// TIA Portal project "2022.10.19_FB_视觉分拣" (V17)
// Vorlageprojekt für das Buch mit Zielsystem S7-1200

(* hardware
DEVICE "S7-1200-Station_1"  S7-1200 Station
   slot 0: "Baugruppenträger_0"  Rack  V1.0
   slot 1: "PLC_1"  CPU 1214C DC/DC/Rly  6ES7 214-1HG40-0XB0  V4.5
*)

// ===== PLC "PLC_1"  CPU 1214C DC/DC/Rly =====

VAR_GLOBAL   // PLC tag table "XML 中的变量表_1"
   "启动按钮" AT %I0.0 : Bool;
   "停止按钮" AT %I0.1 : Bool;
   "复位信号" AT %Q0.2 : Bool;
   "急停" AT %I0.3 : Bool;
   "左电传感器" AT %I0.5 : Bool;
   "后电传感器" AT %I0.7 : Bool;
   "手动模式" AT %I1.0 : Bool;
   "自动模式" AT %I1.1 : Bool;
   "启动指示灯" AT %Q0.0 : Bool;
   "停止指示灯" AT %Q0.1 : Bool;
   "送料带" AT %Q0.3 : Bool;
   "直行电机" AT %Q0.4 : Bool;
   "左换向" AT %Q0.5 : Bool;
   "右换向" AT %Q0.6 : Bool;
   "后1带—原料" AT %Q0.7 : Bool;
   "右1带—基座" AT %Q1.0 : Bool;
   "左1带_产品盖" AT %Q1.1 : Bool;
   "出料台" AT %Q1.2 : Bool;
   "挡板" AT %Q1.3 : Bool;
   "视觉相机" AT %ID30 : DWord;
   "右电传感器" AT %I0.6 : Bool;
END_VAR

DATA_BLOCK "主程序DB"   // DB1
{ S7_Optimized_Access := 'TRUE' }
VERSION : 0.1
   VAR
      核心分拣区程序步 : Int;
   END_VAR
BEGIN
END_DATA_BLOCK

DATA_BLOCK "视觉核心分拣区FB块_DB"   // DB3
{ S7_Optimized_Access := 'TRUE' }
VERSION : 0.1
// stored: InstanceOfName 视觉核心分拣区FB块
"视觉核心分拣区FB块"
BEGIN
END_DATA_BLOCK

FUNCTION_BLOCK "视觉核心分拣区FB块"   // FB1, LAD
{ S7_Optimized_Access := 'TRUE' }
VERSION : 0.1
   VAR_INPUT
      视觉相机数据 : DWord;
      后电传感器 : Bool;
      左电传感器 : Bool;
      右电传感器 : Bool;
   END_VAR
   VAR_OUTPUT
      直行电机 : Bool;
      左转向 : Bool;
      右转向 : Bool;
   END_VAR
   VAR_IN_OUT
      程序步 : Int;
   END_VAR
   VAR
      中间变量1 : Bool;
      中间变量2 : Bool;
      中间变量3 : Bool;
   END_VAR
   VAR_TEMP   // added for the SCL form of the ladder/FBD networks
      _w1 : Bool;
   END_VAR
BEGIN

REGION Network 1: 物料判断
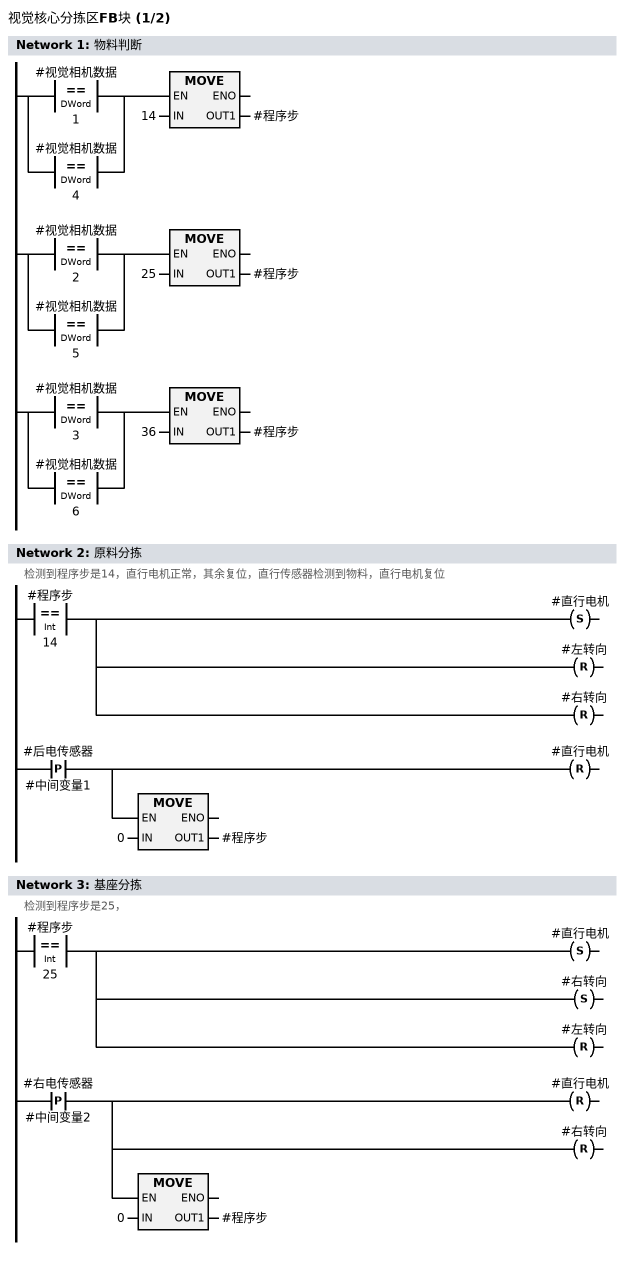
   RUNG wire#powerrail
      { S7_Templates := "SrcType := DWord" } EQ_Contact(in1 := #视觉相机数据, in2 := 1)
      wire#w1
      Move(in := 14, out1 => #程序步)
   END_RUNG
   RUNG wire#powerrail
      { S7_Templates := "SrcType := DWord" } EQ_Contact(in1 := #视觉相机数据, in2 := 4)
   END_RUNG wire#w1
   RUNG wire#powerrail
      { S7_Templates := "SrcType := DWord" } EQ_Contact(in1 := #视觉相机数据, in2 := 2)
      wire#w2
      Move(in := 25, out1 => #程序步)
   END_RUNG
   RUNG wire#powerrail
      { S7_Templates := "SrcType := DWord" } EQ_Contact(in1 := #视觉相机数据, in2 := 5)
   END_RUNG wire#w2
   RUNG wire#powerrail
      { S7_Templates := "SrcType := DWord" } EQ_Contact(in1 := #视觉相机数据, in2 := 3)
      wire#w3
      Move(in := 36, out1 => #程序步)
   END_RUNG
   RUNG wire#powerrail
      { S7_Templates := "SrcType := DWord" } EQ_Contact(in1 := #视觉相机数据, in2 := 6)
   END_RUNG wire#w3
   // the same network as SCL:
   IF (#视觉相机数据 = 1) OR (#视觉相机数据 = 4) THEN #程序步 := 14; END_IF;
   IF (#视觉相机数据 = 2) OR (#视觉相机数据 = 5) THEN #程序步 := 25; END_IF;
   IF (#视觉相机数据 = 3) OR (#视觉相机数据 = 6) THEN #程序步 := 36; END_IF;
END_REGION

REGION Network 2: 原料分拣
   // 检测到程序步是14，直行电机正常，其余复位，直行传感器检测到物料，直行电机复位
   RUNG wire#powerrail
      { S7_Templates := "SrcType := Int" } EQ_Contact(in1 := #程序步, in2 := 14)
      wire#w1
      S_Coil( #直行电机 )
   END_RUNG
   RUNG wire#w1
      R_Coil( #左转向 )
   END_RUNG
   RUNG wire#w1
      R_Coil( #右转向 )
   END_RUNG
   RUNG wire#powerrail
      P_Contact(operand := #后电传感器, bit := #中间变量1)
      wire#w2
      R_Coil( #直行电机 )
   END_RUNG
   RUNG wire#w2
      Move(in := 0, out1 => #程序步)
   END_RUNG
   // the same network as SCL:
   IF #程序步 = 14 THEN
       #直行电机 := TRUE;
       #左转向 := FALSE;
       #右转向 := FALSE;
   END_IF;
   #_w1 := #后电传感器 AND NOT #中间变量1;   // rising edge of #后电传感器
   #中间变量1 := #后电传感器;
   IF #_w1 THEN
       #直行电机 := FALSE;
       #程序步 := 0;
   END_IF;
END_REGION

REGION Network 3: 基座分拣
   // 检测到程序步是25，
   RUNG wire#powerrail
      { S7_Templates := "SrcType := Int" } EQ_Contact(in1 := #程序步, in2 := 25)
      wire#w1
      S_Coil( #直行电机 )
   END_RUNG
   RUNG wire#w1
      S_Coil( #右转向 )
   END_RUNG
   RUNG wire#w1
      R_Coil( #左转向 )
   END_RUNG
   RUNG wire#powerrail
      P_Contact(operand := #右电传感器, bit := #中间变量2)
      wire#w2
      R_Coil( #直行电机 )
   END_RUNG
   RUNG wire#w2
      R_Coil( #右转向 )
   END_RUNG
   RUNG wire#w2
      Move(in := 0, out1 => #程序步)
   END_RUNG
   // the same network as SCL:
   IF #程序步 = 25 THEN
       #直行电机 := TRUE;
       #右转向 := TRUE;
       #左转向 := FALSE;
   END_IF;
   #_w1 := #右电传感器 AND NOT #中间变量2;   // rising edge of #右电传感器
   #中间变量2 := #右电传感器;
   IF #_w1 THEN
       #直行电机 := FALSE;
       #右转向 := FALSE;
       #程序步 := 0;
   END_IF;
END_REGION

REGION Network 4: 基盖
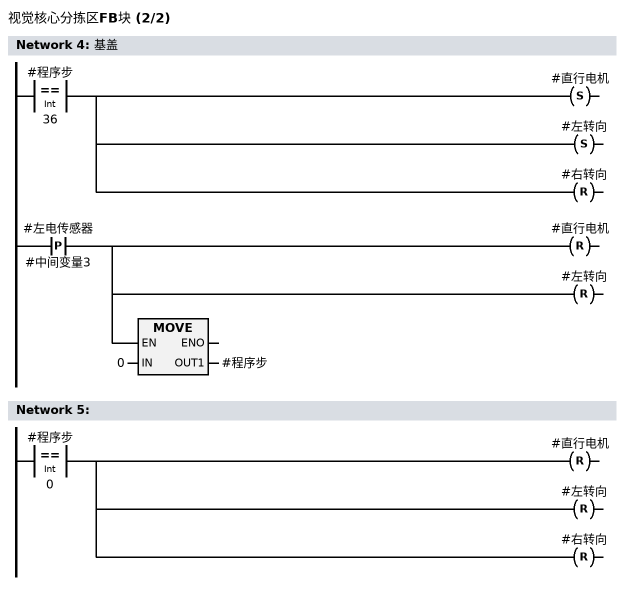
   RUNG wire#powerrail
      { S7_Templates := "SrcType := Int" } EQ_Contact(in1 := #程序步, in2 := 36)
      wire#w1
      S_Coil( #直行电机 )
   END_RUNG
   RUNG wire#w1
      S_Coil( #左转向 )
   END_RUNG
   RUNG wire#w1
      R_Coil( #右转向 )
   END_RUNG
   RUNG wire#powerrail
      P_Contact(operand := #左电传感器, bit := #中间变量3)
      wire#w2
      R_Coil( #直行电机 )
   END_RUNG
   RUNG wire#w2
      R_Coil( #左转向 )
   END_RUNG
   RUNG wire#w2
      Move(in := 0, out1 => #程序步)
   END_RUNG
   // the same network as SCL:
   IF #程序步 = 36 THEN
       #直行电机 := TRUE;
       #左转向 := TRUE;
       #右转向 := FALSE;
   END_IF;
   #_w1 := #左电传感器 AND NOT #中间变量3;   // rising edge of #左电传感器
   #中间变量3 := #左电传感器;
   IF #_w1 THEN
       #直行电机 := FALSE;
       #左转向 := FALSE;
       #程序步 := 0;
   END_IF;
END_REGION

REGION Network 5
   RUNG wire#powerrail
      { S7_Templates := "SrcType := Int" } EQ_Contact(in1 := #程序步, in2 := 0)
      wire#w1
      R_Coil( #直行电机 )
   END_RUNG
   RUNG wire#w1
      R_Coil( #左转向 )
   END_RUNG
   RUNG wire#w1
      R_Coil( #右转向 )
   END_RUNG
   // the same network as SCL:
   IF #程序步 = 0 THEN
       #直行电机 := FALSE;
       #左转向 := FALSE;
       #右转向 := FALSE;
   END_IF;
END_REGION
END_FUNCTION_BLOCK

FUNCTION "MHJ-PLC-Lab-Function-S71200" : Void   // FC9000, SCL
{ S7_Optimized_Access := 'TRUE' }
VERSION : 0.1
   VAR_TEMP
      rdTimeReturn : Int;
      outputTime : DTL;
      SyncVal : Byte;
      forVal : Int;
      forVal_2 : Int;
      Value : Byte;
   END_VAR
   VAR CONSTANT
      CompVal : Byte := 16#34;
      Value_01 : Byte := 16#11;
      Value_01_DW : DWord := 16#A165_D992;
      Value_02_DW : DWord := 16#58BE_4401;
   END_VAR
BEGIN

   #Value:=PEEK(area := 16#82,
        dbNumber := 0,
        byteOffset := 511);
   #Value := #Value + 1;

   POKE(area := 16#82,
        dbNumber := 0,
        byteOffset := 511,
        value := #Value);

   POKE(area:=16#81,
        dbNumber:=0,
        byteOffset:=1016,
        value:=#Value_01_DW);
   POKE(area := 16#81,
        dbNumber := 0,
        byteOffset := 1020,
        value := #Value_02_DW);

   POKE(area := 16#81,
        dbNumber := 0,
        byteOffset := 511,
        value := B#16#00);

   FOR #forVal := 0 TO 120 DO
       FOR #forVal_2:=0 TO 10 DO
           #rdTimeReturn:=RD_SYS_T(#outputTime);
           #rdTimeReturn := WR_SYS_T(#outputTime);
           #rdTimeReturn := RD_SYS_T(#outputTime);
           #rdTimeReturn := WR_SYS_T(#outputTime);
       END_FOR;
       #SyncVal:= PEEK(area := 16#81,
                      dbNumber := 0,
                      byteOffset := 511);
       IF #SyncVal = #CompVal THEN
          GOTO M_1;
       END_IF;
   END_FOR;
   RETURN;

   M_1:
   POKE(area := 16#81,
        dbNumber := 0,
        byteOffset := 511,
        value := B#16#0);
END_FUNCTION

ORGANIZATION_BLOCK "Main"   // OB1, LAD, ProgramCycle
TITLE = "Main Program Sweep (Cycle)"
{ S7_Optimized_Access := 'TRUE' }
VERSION : 0.1
   VAR_INPUT
      Initial_Call : Bool;   // Initial call of this OB
      Remanence : Bool;   // =True, if remanent data are available
   END_VAR
BEGIN

REGION Network 1: Konnektierungsbaustein für PLC-Lab
   // Im Netzwerk 1 wird der Konnektierungsbaustein für PLC-Lab aufgerufen.
   // Dieser Aufruf darf nicht entfernt werden!
   // Factory_调试按钮时，需要人工触发的一开始点开，亮成闪电状，需要触发的调成没有故障，白色小眼睛
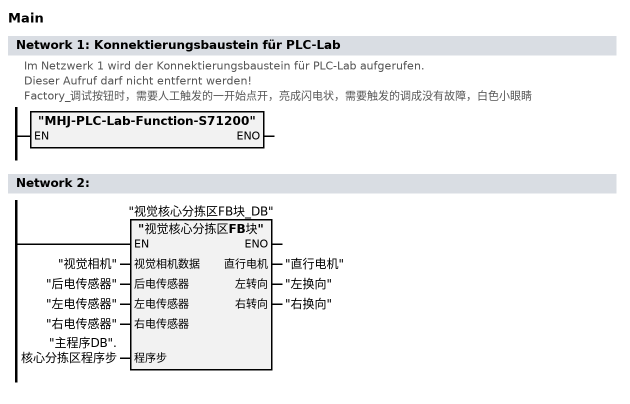
   RUNG wire#powerrail
      "MHJ-PLC-Lab-Function-S71200"()
   END_RUNG
   // the same network as SCL:
   "MHJ-PLC-Lab-Function-S71200"();
END_REGION

REGION Network 2
   RUNG wire#powerrail
      "视觉核心分拣区FB块_DB"(视觉相机数据 := "视觉相机", 后电传感器 := "后电传感器", 左电传感器 := "左电传感器", 右电传感器 := "右电传感器", 程序步 := "主程序DB".核心分拣区程序步, 直行电机 => "直行电机", 左转向 => "左换向", 右转向 => "右换向")
   END_RUNG
   // the same network as SCL:
   "视觉核心分拣区FB块_DB"(视觉相机数据 := "视觉相机",   // "视觉核心分拣区FB块"
                   后电传感器 := "后电传感器",
                   左电传感器 := "左电传感器",
                   右电传感器 := "右电传感器",
                   程序步 := "主程序DB".核心分拣区程序步,
                   直行电机 => "直行电机",
                   左转向 => "左换向",
                   右转向 => "右换向");
END_REGION
END_ORGANIZATION_BLOCK